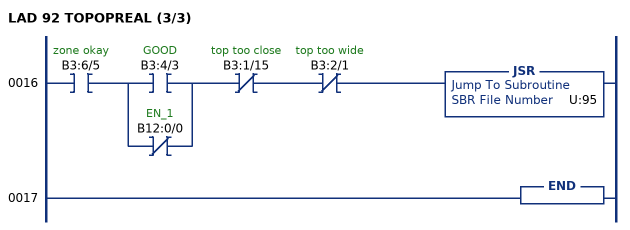
% Rung: 16 %
SOR XIC B3:6/5 BST XIC B3:4/3 NXB XIO B12:0/0 BND XIO B3:1/15 XIO B3:2/1 JSR U:95 EOR
%   B3:6/5  "zone okay" %
%   B3:4/3  GOOD %
%   B12:0/0  EN_1 %
%   B3:1/15  "top too close" %
%   B3:2/1  "top too wide" %
% Rung: 17 %
SOR END EOR

LADDER 93 "TOPOPTEST"
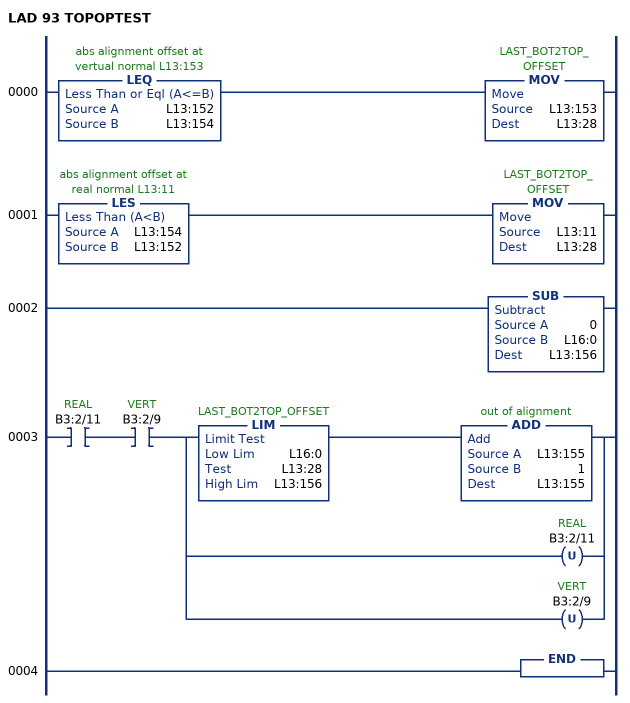
% Rung: 0 %
SOR LEQ L13:152 L13:154 MOV L13:153 L13:28 EOR
%   L13:152  "abs alignment offset at vertual normal L13:153" %
%   L13:154  "abs alignment offset at real normal L13:11" %
%   L13:153  "normal alignment offset at vertual abs L13:152" %
%   L13:28  LAST_BOT2TOP_OFFSET %
% Rung: 1 %
SOR LES L13:154 L13:152 MOV L13:11 L13:28 EOR
%   L13:154  "abs alignment offset at real normal L13:11" %
%   L13:152  "abs alignment offset at vertual normal L13:153" %
%   L13:11  "normal alignment offset at real abs L13:154" %
%   L13:28  LAST_BOT2TOP_OFFSET %
% Rung: 2 %
SOR SUB 0 L16:0 L13:156 EOR
%   L16:0  MAX_OFFSET %
% Rung: 3 %
SOR XIC B3:2/11 XIC B3:2/9 BST LIM L16:0 L13:28 L13:156 ADD L13:155 1 L13:155 NXB OTU B3:2/11 NXB OTU B3:2/9 BND EOR
%   B3:2/11  REAL %
%   B3:2/9  VERT %
%   L16:0  MAX_OFFSET %
%   L13:28  LAST_BOT2TOP_OFFSET %
%   L13:155  "out of alignment" %
% Rung: 4 %
SOR END EOR

LADDER 94 "TOPOPRANGE"
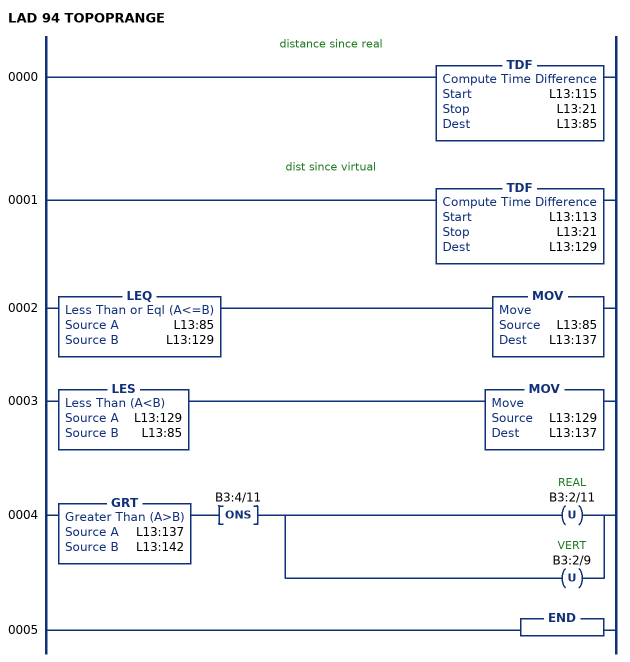
% Rung: 0 %
% distance since real %
SOR TDF L13:115 L13:21 L13:85 EOR
%   L13:115  TRAILING_EDGE_RAW  "top optic trailing edge position" %
%   L13:21  TOP_POSITION %
% Rung: 1 %
% dist since virtual %
SOR TDF L13:113 L13:21 L13:129 EOR
%   L13:113  VERTUAL_PT_RAW_CL  "virtual part center line transfer from the bottom in raw position" %
%   L13:21  TOP_POSITION %
% Rung: 2 %
SOR LEQ L13:85 L13:129 MOV L13:85 L13:137 EOR
% Rung: 3 %
SOR LES L13:129 L13:85 MOV L13:129 L13:137 EOR
% Rung: 4 %
SOR GRT L13:137 L13:142 ONS B3:4/11 BST OTU B3:2/11 NXB OTU B3:2/9 BND EOR
%   L13:142  LAST_ALIGNMENT_FAILS %
%   B3:2/11  REAL %
%   B3:2/9  VERT %
% Rung: 5 %
SOR END EOR

LADDER 95 "TOPOPOKAY"
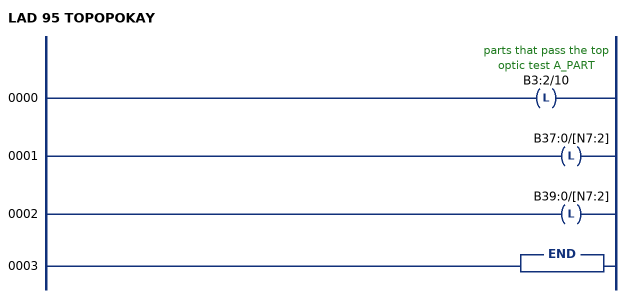
% Rung: 0 %
SOR OTL B3:2/10 EOR
%   B3:2/10  A_PART  "parts that pass the top optic test" %
% Rung: 1 %
SOR OTL B37:0/[N7:2] EOR
%   B37:0  TOP_GOOD %
%   N7:2  TOP_OPTIC_LOAD_LOC  "part load location" %
% Rung: 2 %
SOR OTL B39:0/[N7:2] EOR
%   B39:0  EX2_GOOD %
%   N7:2  TOP_OPTIC_LOAD_LOC  "part load location" %
% Rung: 3 %
SOR END EOR

LADDER 100 "1 INS5"
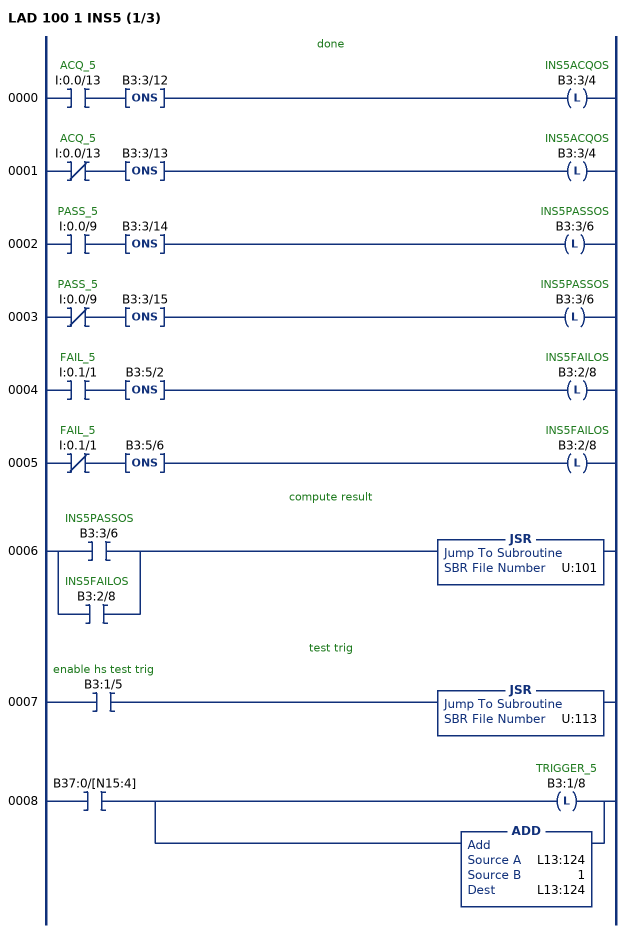
% Rung: 0 %
% done %
SOR XIC I:0.0/13 ONS B3:3/12 OTL B3:3/4 EOR
%   I:0.0/13  ACQ_5 %
%   B3:3/4  INS5ACQOS %
% Rung: 1 %
SOR XIO I:0.0/13 ONS B3:3/13 OTL B3:3/4 EOR
%   I:0.0/13  ACQ_5 %
%   B3:3/4  INS5ACQOS %
% Rung: 2 %
SOR XIC I:0.0/9 ONS B3:3/14 OTL B3:3/6 EOR
%   I:0.0/9  PASS_5 %
%   B3:3/6  INS5PASSOS %
% Rung: 3 %
SOR XIO I:0.0/9 ONS B3:3/15 OTL B3:3/6 EOR
%   I:0.0/9  PASS_5 %
%   B3:3/6  INS5PASSOS %
% Rung: 4 %
SOR XIC I:0.1/1 ONS B3:5/2 OTL B3:2/8 EOR
%   I:0.1/1  FAIL_5 %
%   B3:2/8  INS5FAILOS %
% Rung: 5 %
SOR XIO I:0.1/1 ONS B3:5/6 OTL B3:2/8 EOR
%   I:0.1/1  FAIL_5 %
%   B3:2/8  INS5FAILOS %
% Rung: 6 %
% compute result %
SOR BST XIC B3:3/6 NXB XIC B3:2/8 BND JSR U:101 EOR
%   B3:3/6  INS5PASSOS %
%   B3:2/8  INS5FAILOS %
% Rung: 7 %
% test trig %
SOR XIC B3:1/5 JSR U:113 EOR
%   B3:1/5  "enable hs test trig" %
% Rung: 8 %
SOR XIC B37:0/[N15:4] BST OTL B3:1/8 NXB ADD L13:124 1 L13:124 BND EOR
%   B37:0  TOP_GOOD %
%   N15:4  INS_5_TRIG_LOC %
%   B3:1/8  TRIGGER_5 %

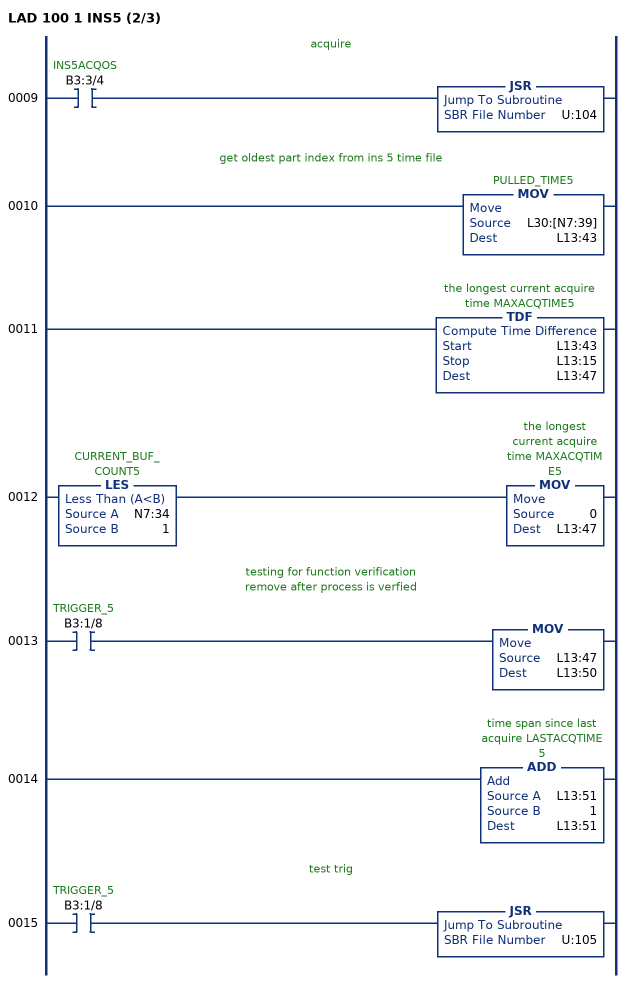
% Rung: 9 %
% acquire %
SOR XIC B3:3/4 JSR U:104 EOR
%   B3:3/4  INS5ACQOS %
% Rung: 10 %
% get oldest part index from ins 5 time file %
SOR MOV L30:[N7:39] L13:43 EOR
%   N7:39  OLDEST_PART_INDEX5 %
%   L13:43  PULLED_TIME5 %
% Rung: 11 %
SOR TDF L13:43 L13:15 L13:47 EOR
%   L13:43  PULLED_TIME5 %
%   L13:15  THE_TIME %
%   L13:47  MAXACQTIME5  "the longest current acquire time" %
% Rung: 12 %
SOR LES N7:34 1 MOV 0 L13:47 EOR
%   N7:34  CURRENT_BUF_COUNT5 %
%   L13:47  MAXACQTIME5  "the longest current acquire time" %
% Rung: 13 %
% testing for function verification
% remove after process is verfied %
SOR XIC B3:1/8 MOV L13:47 L13:50 EOR
%   B3:1/8  TRIGGER_5 %
%   L13:47  MAXACQTIME5  "the longest current acquire time" %
% Rung: 14 %
SOR ADD L13:51 1 L13:51 EOR
%   L13:51  LASTACQTIME5  "time span since last acquire" %
% Rung: 15 %
% test trig %
SOR XIC B3:1/8 JSR U:105 EOR
%   B3:1/8  TRIGGER_5 %

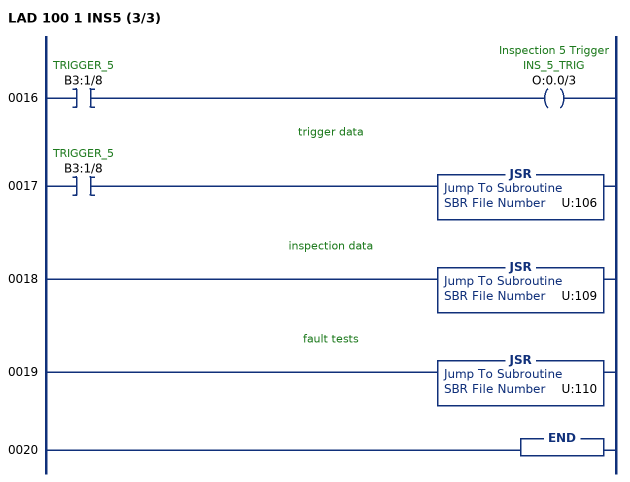
% Rung: 16 %
SOR XIC B3:1/8 OTE O:0.0/3 EOR
%   B3:1/8  TRIGGER_5 %
%   O:0.0/3  INS_5_TRIG  "Inspection 5 Trigger" %
% Rung: 17 %
% trigger data %
SOR XIC B3:1/8 JSR U:106 EOR
%   B3:1/8  TRIGGER_5 %
% Rung: 18 %
% inspection data %
SOR JSR U:109 EOR
% Rung: 19 %
% fault tests %
SOR JSR U:110 EOR
% Rung: 20 %
SOR END EOR

LADDER 101 "2 INS5RESU"
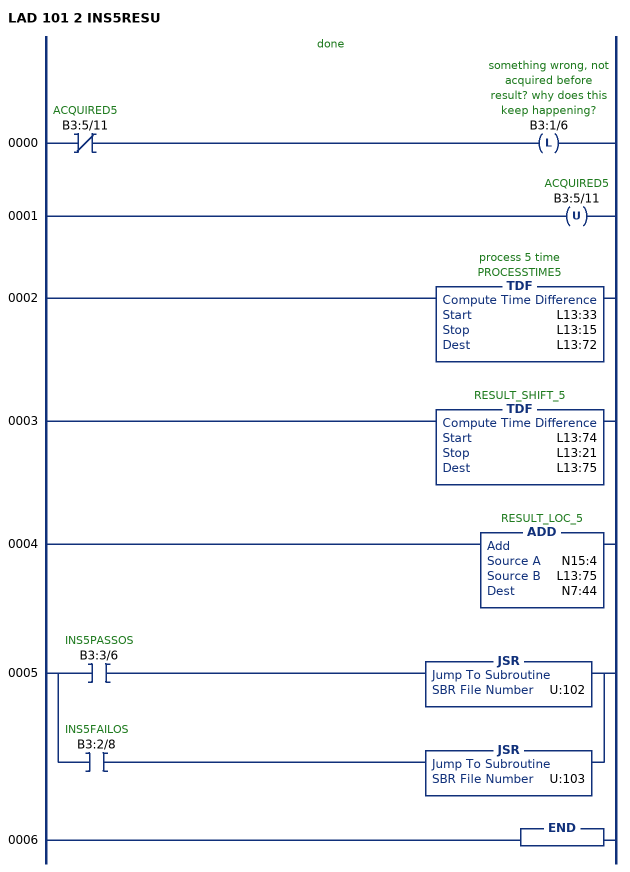
% Rung: 0 %
% done %
SOR XIO B3:5/11 OTL B3:1/6 EOR
%   B3:5/11  ACQUIRED5 %
%   B3:1/6  "something wrong, not acquired before result? why does this keep happening?" %
% Rung: 1 %
SOR OTU B3:5/11 EOR
%   B3:5/11  ACQUIRED5 %
% Rung: 2 %
SOR TDF L13:33 L13:15 L13:72 EOR
%   L13:33  TIMEOFACQ5  "the time of the last acquire" %
%   L13:15  THE_TIME %
%   L13:72  PROCESSTIME5  "process 5 time" %
% Rung: 3 %
SOR TDF L13:74 L13:21 L13:75 EOR
%   L13:74  PROCESS_START_POS_5 %
%   L13:21  TOP_POSITION %
%   L13:75  RESULT_SHIFT_5 %
% Rung: 4 %
SOR ADD N15:4 L13:75 N7:44 EOR
%   N15:4  INS_5_TRIG_LOC %
%   L13:75  RESULT_SHIFT_5 %
%   N7:44  RESULT_LOC_5 %
% Rung: 5 %
SOR BST XIC B3:3/6 JSR U:102 NXB XIC B3:2/8 JSR U:103 BND EOR
%   B3:3/6  INS5PASSOS %
%   B3:2/8  INS5FAILOS %
% Rung: 6 %
SOR END EOR

LADDER 102 "3 INS5PASS"
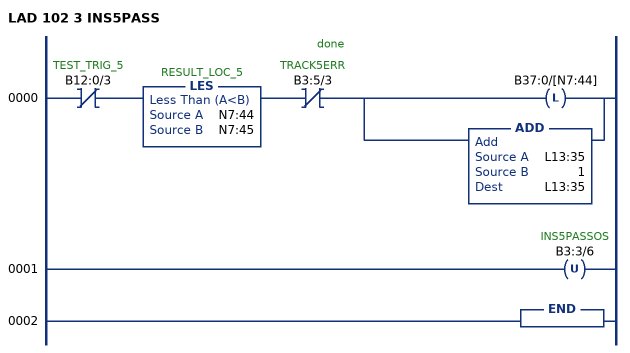
% Rung: 0 %
% done %
SOR XIO B12:0/3 LES N7:44 N7:45 XIO B3:5/3 BST OTL B37:0/[N7:44] NXB ADD L13:35 1 L13:35 BND EOR
%   B12:0/3  TEST_TRIG_5 %
%   N7:44  RESULT_LOC_5 %
%   N7:45  INS5_MAX_SHIFT  "ins 5 maximum result location" %
%   B3:5/3  TRACK5ERR %
%   B37:0  TOP_GOOD %
% Rung: 1 %
SOR OTU B3:3/6 EOR
%   B3:3/6  INS5PASSOS %
% Rung: 2 %
SOR END EOR

LADDER 103 "4 INS5FAIL"
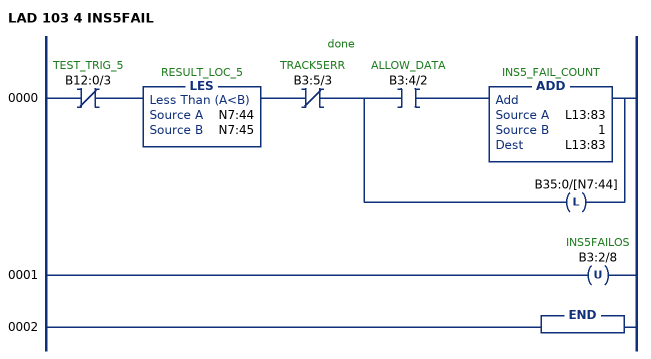
% Rung: 0 %
% done %
SOR XIO B12:0/3 LES N7:44 N7:45 XIO B3:5/3 BST XIC B3:4/2 ADD L13:83 1 L13:83 NXB OTL B35:0/[N7:44] BND EOR
%   B12:0/3  TEST_TRIG_5 %
%   N7:44  RESULT_LOC_5 %
%   N7:45  INS5_MAX_SHIFT  "ins 5 maximum result location" %
%   B3:5/3  TRACK5ERR %
%   B3:4/2  ALLOW_DATA %
%   L13:83  INS5_FAIL_COUNT %
%   B35:0  TOP_NG %
% Rung: 1 %
SOR OTU B3:2/8 EOR
%   B3:2/8  INS5FAILOS %
% Rung: 2 %
SOR END EOR

LADDER 104 "5 INS5ACQ"
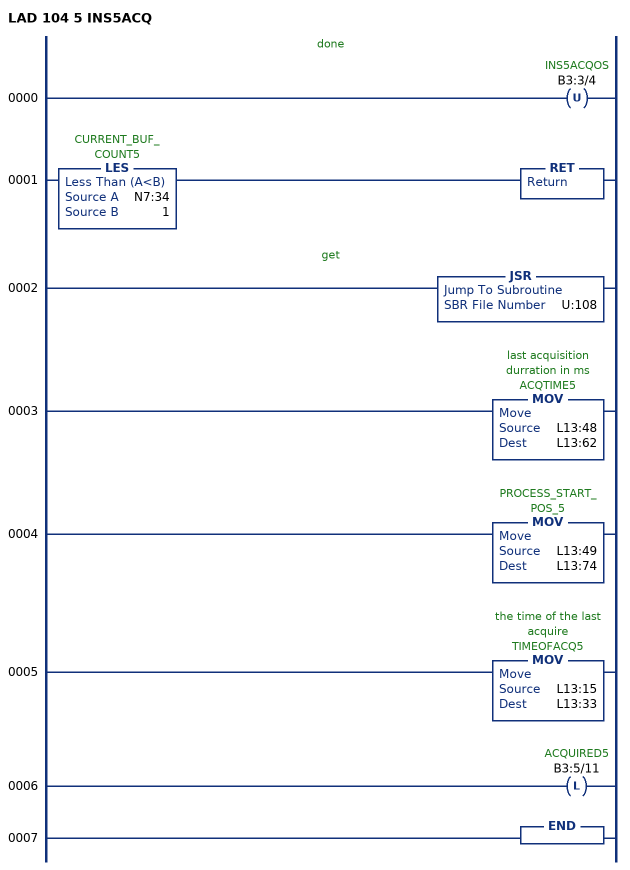
% Rung: 0 %
% done %
SOR OTU B3:3/4 EOR
%   B3:3/4  INS5ACQOS %
% Rung: 1 %
SOR LES N7:34 1 RET EOR
%   N7:34  CURRENT_BUF_COUNT5 %
% Rung: 2 %
% get %
SOR JSR U:108 EOR
% Rung: 3 %
SOR MOV L13:48 L13:62 EOR
%   L13:48  TIME_SPAN5 %
%   L13:62  ACQTIME5  "last acquisition durration in ms" %
% Rung: 4 %
SOR MOV L13:49 L13:74 EOR
%   L13:49  PULLED_POSITION5 %
%   L13:74  PROCESS_START_POS_5 %
% Rung: 5 %
SOR MOV L13:15 L13:33 EOR
%   L13:15  THE_TIME %
%   L13:33  TIMEOFACQ5  "the time of the last acquire" %
% Rung: 6 %
SOR OTL B3:5/11 EOR
%   B3:5/11  ACQUIRED5 %
% Rung: 7 %
SOR END EOR

LADDER 105 "6 Q5TESTTR"
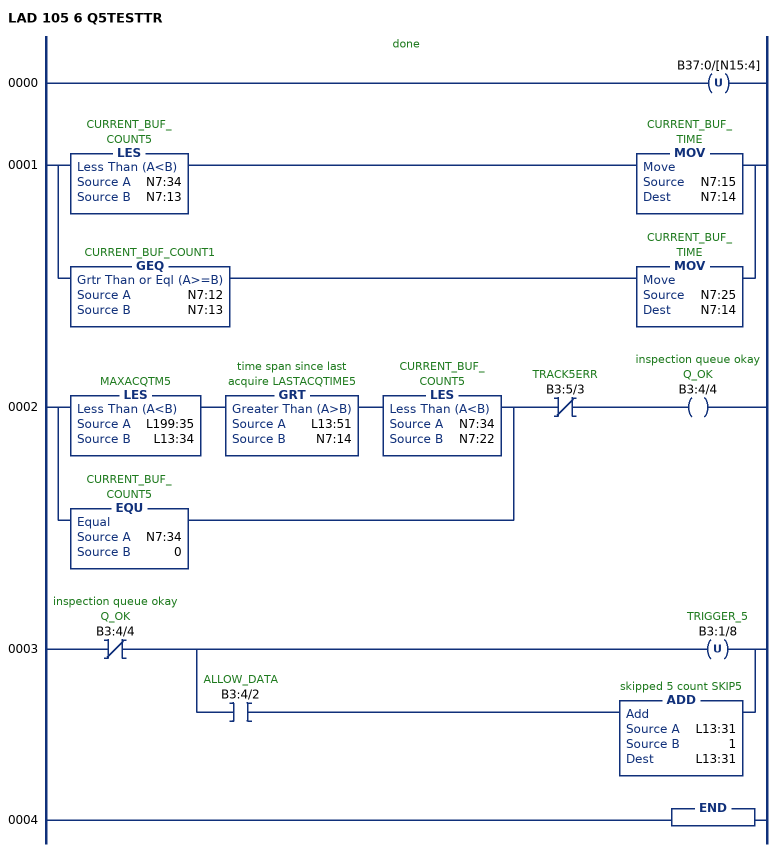
% Rung: 0 %
% done %
SOR OTU B37:0/[N15:4] EOR
%   B37:0  TOP_GOOD %
%   N15:4  INS_5_TRIG_LOC %
% Rung: 1 %
SOR BST LES N7:34 N7:13 MOV N7:15 N7:14 NXB GEQ N7:12 N7:13 MOV N7:25 N7:14 BND EOR
%   N7:34  CURRENT_BUF_COUNT5 %
%   N7:13  BUF_TRANS  "cam to pc buf transition" %
%   N7:15  CAM_BUF_TIME  "cam buf time" %
%   N7:14  CURRENT_BUF_TIME %
%   N7:12  CURRENT_BUF_COUNT1 %
%   N7:25  PC_BUF_TIME  "pc buf time" %
% Rung: 2 %
SOR BST LES L199:35 L13:34 GRT L13:51 N7:14 LES N7:34 N7:22 NXB EQU N7:34 0 BND XIO B3:5/3 OTE B3:4/4 EOR
%   L199:35  MAXACQTM5 %
%   L13:34  MAX_ACQ_ALL  "absolute max acquire time before bypass trigger" %
%   L13:51  LASTACQTIME5  "time span since last acquire" %
%   N7:14  CURRENT_BUF_TIME %
%   N7:34  CURRENT_BUF_COUNT5 %
%   N7:22  MAX_BUF_ALL  "max buffer count alowed before bypass" %
%   B3:5/3  TRACK5ERR %
%   B3:4/4  Q_OK  "inspection queue okay" %
% Rung: 3 %
SOR XIO B3:4/4 BST OTU B3:1/8 NXB XIC B3:4/2 ADD L13:31 1 L13:31 BND EOR
%   B3:4/4  Q_OK  "inspection queue okay" %
%   B3:1/8  TRIGGER_5 %
%   B3:4/2  ALLOW_DATA %
%   L13:31  SKIP5  "skipped 5 count" %
% Rung: 4 %
SOR END EOR

LADDER 106 "7 INS5TRIG"
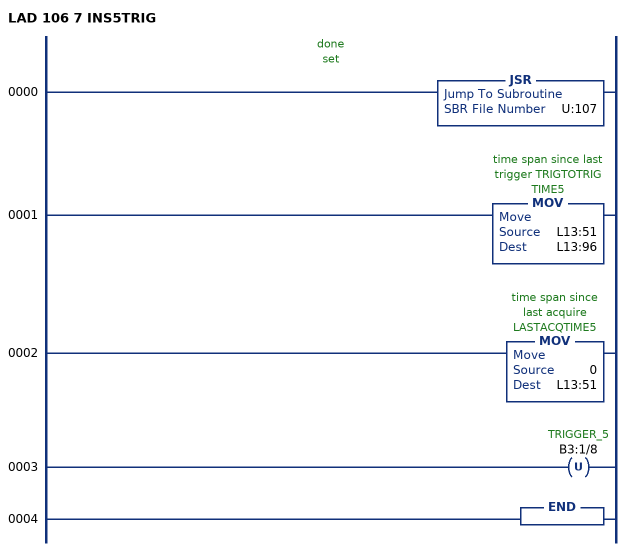
% Rung: 0 %
% done
% set %
SOR JSR U:107 EOR
% Rung: 1 %
SOR MOV L13:51 L13:96 EOR
%   L13:51  LASTACQTIME5  "time span since last acquire" %
%   L13:96  TRIGTOTRIGTIME5  "time span since last trigger" %
% Rung: 2 %
SOR MOV 0 L13:51 EOR
%   L13:51  LASTACQTIME5  "time span since last acquire" %
% Rung: 3 %
SOR OTU B3:1/8 EOR
%   B3:1/8  TRIGGER_5 %
% Rung: 4 %
SOR END EOR

LADDER 107 "8 FIFO5SET"
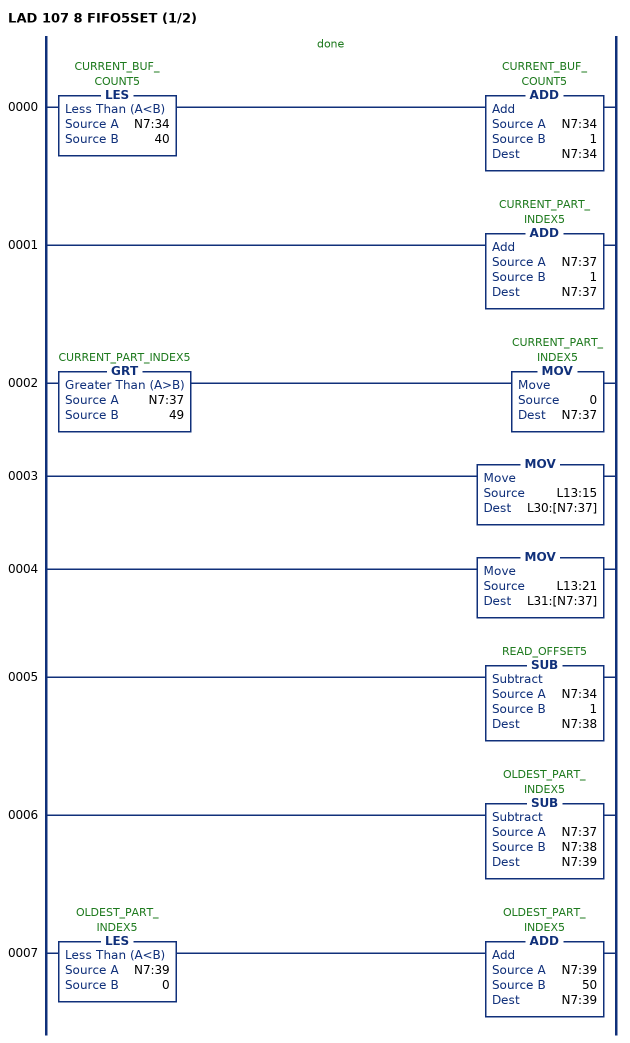
% Rung: 0 %
% done %
SOR LES N7:34 40 ADD N7:34 1 N7:34 EOR
%   N7:34  CURRENT_BUF_COUNT5 %
% Rung: 1 %
SOR ADD N7:37 1 N7:37 EOR
%   N7:37  CURRENT_PART_INDEX5 %
% Rung: 2 %
SOR GRT N7:37 49 MOV 0 N7:37 EOR
%   N7:37  CURRENT_PART_INDEX5 %
% Rung: 3 %
SOR MOV L13:15 L30:[N7:37] EOR
%   L13:15  THE_TIME %
%   N7:37  CURRENT_PART_INDEX5 %
% Rung: 4 %
SOR MOV L13:21 L31:[N7:37] EOR
%   L13:21  TOP_POSITION %
%   N7:37  CURRENT_PART_INDEX5 %
% Rung: 5 %
SOR SUB N7:34 1 N7:38 EOR
%   N7:34  CURRENT_BUF_COUNT5 %
%   N7:38  READ_OFFSET5 %
% Rung: 6 %
SOR SUB N7:37 N7:38 N7:39 EOR
%   N7:37  CURRENT_PART_INDEX5 %
%   N7:38  READ_OFFSET5 %
%   N7:39  OLDEST_PART_INDEX5 %
% Rung: 7 %
SOR LES N7:39 0 ADD N7:39 50 N7:39 EOR
%   N7:39  OLDEST_PART_INDEX5 %

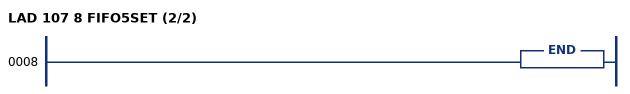
% Rung: 8 %
SOR END EOR

LADDER 108 "9 FIFO5GET"
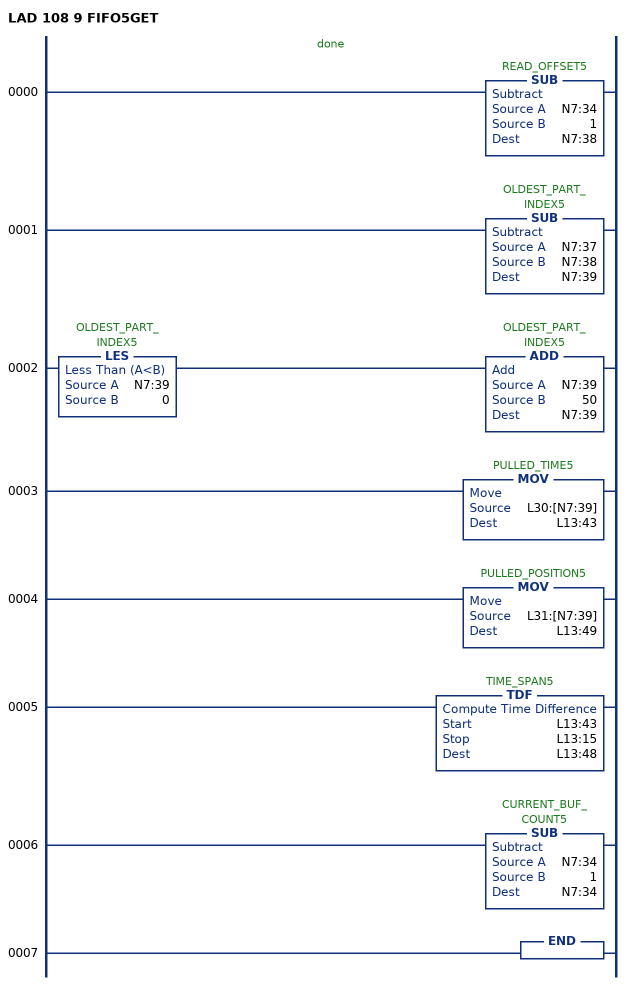
% Rung: 0 %
% done %
SOR SUB N7:34 1 N7:38 EOR
%   N7:34  CURRENT_BUF_COUNT5 %
%   N7:38  READ_OFFSET5 %
% Rung: 1 %
SOR SUB N7:37 N7:38 N7:39 EOR
%   N7:37  CURRENT_PART_INDEX5 %
%   N7:38  READ_OFFSET5 %
%   N7:39  OLDEST_PART_INDEX5 %
% Rung: 2 %
SOR LES N7:39 0 ADD N7:39 50 N7:39 EOR
%   N7:39  OLDEST_PART_INDEX5 %
% Rung: 3 %
SOR MOV L30:[N7:39] L13:43 EOR
%   N7:39  OLDEST_PART_INDEX5 %
%   L13:43  PULLED_TIME5 %
% Rung: 4 %
SOR MOV L31:[N7:39] L13:49 EOR
%   N7:39  OLDEST_PART_INDEX5 %
%   L13:49  PULLED_POSITION5 %
% Rung: 5 %
SOR TDF L13:43 L13:15 L13:48 EOR
%   L13:43  PULLED_TIME5 %
%   L13:15  THE_TIME %
%   L13:48  TIME_SPAN5 %
% Rung: 6 %
SOR SUB N7:34 1 N7:34 EOR
%   N7:34  CURRENT_BUF_COUNT5 %
% Rung: 7 %
SOR END EOR

LADDER 109 "10INSDATA5"
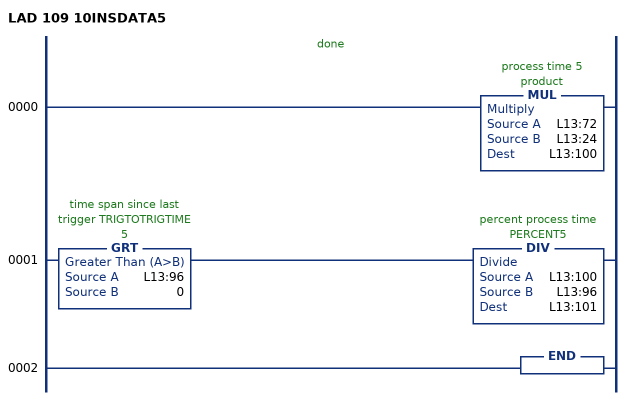
% Rung: 0 %
% done %
SOR MUL L13:72 L13:24 L13:100 EOR
%   L13:72  PROCESSTIME5  "process 5 time" %
%   L13:24  "multiplyer to make devision come out to a percentage" %
%   L13:100  "process time 5 product" %
% Rung: 1 %
SOR GRT L13:96 0 DIV L13:100 L13:96 L13:101 EOR
%   L13:96  TRIGTOTRIGTIME5  "time span since last trigger" %
%   L13:100  "process time 5 product" %
%   L13:101  PERCENT5  "percent process time" %
% Rung: 2 %
SOR END EOR

LADDER 110 "11TSTFALT5"
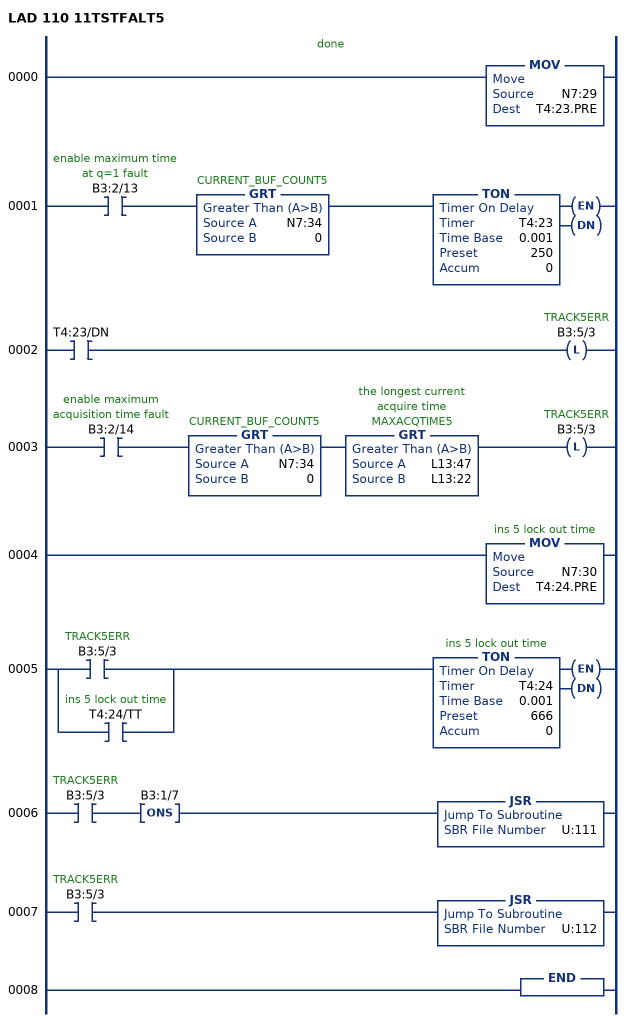
% Rung: 0 %
% done %
SOR MOV N7:29 T4:23.PRE EOR
%   N7:29  "max allowed ms time for q to be above 1 if safe fault is used" %
% Rung: 1 %
SOR XIC B3:2/13 GRT N7:34 0 TON T4:23 0.001 250 0 EOR
%   B3:2/13  "enable maximum time at q=1 fault" %
%   N7:34  CURRENT_BUF_COUNT5 %
% Rung: 2 %
SOR XIC T4:23/DN OTL B3:5/3 EOR
%   B3:5/3  TRACK5ERR %
% Rung: 3 %
SOR XIC B3:2/14 GRT N7:34 0 GRT L13:47 L13:22 OTL B3:5/3 EOR
%   B3:2/14  "enable maximum acquisition time fault" %
%   N7:34  CURRENT_BUF_COUNT5 %
%   L13:47  MAXACQTIME5  "the longest current acquire time" %
%   L13:22  "maximum of the longest acquire time allowed if maximum acquire time fault is enabled" %
%   B3:5/3  TRACK5ERR %
% Rung: 4 %
SOR MOV N7:30 T4:24.PRE EOR
%   N7:30  "ms time setting to lock out inspection to give all pending images a chance to clear" %
%   T4:24  "ins 5 lock out time" %
% Rung: 5 %
SOR BST XIC B3:5/3 NXB XIC T4:24/TT BND TON T4:24 0.001 666 0 EOR
%   B3:5/3  TRACK5ERR %
%   T4:24  "ins 5 lock out time" %
% Rung: 6 %
SOR XIC B3:5/3 ONS B3:1/7 JSR U:111 EOR
%   B3:5/3  TRACK5ERR %
% Rung: 7 %
SOR XIC B3:5/3 JSR U:112 EOR
%   B3:5/3  TRACK5ERR %
% Rung: 8 %
SOR END EOR

LADDER 111 "12INS5FIX1"
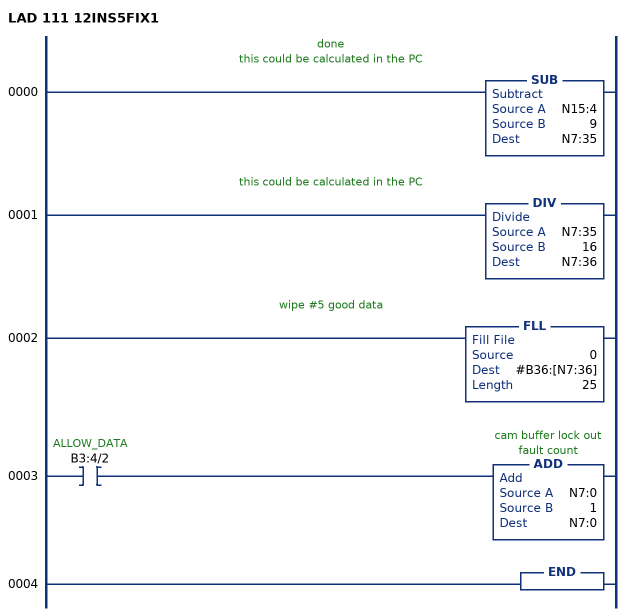
% Rung: 0 %
% done
% this could be calculated in the PC %
SOR SUB N15:4 9 N7:35 EOR
%   N15:4  INS_5_TRIG_LOC %
% Rung: 1 %
% this could be calculated in the PC %
SOR DIV N7:35 16 N7:36 EOR
% Rung: 2 %
% wipe #5 good data %
SOR FLL 0 #B36:[N7:36] 25 EOR
% Rung: 3 %
SOR XIC B3:4/2 ADD N7:0 1 N7:0 EOR
%   B3:4/2  ALLOW_DATA %
%   N7:0  "cam buffer lock out fault count" %
% Rung: 4 %
SOR END EOR

LADDER 112 "13INS5FIX2"
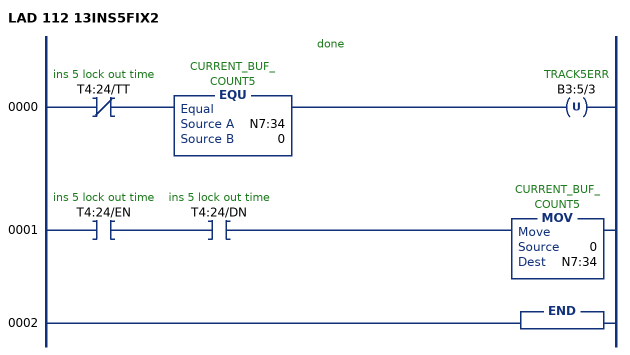
% Rung: 0 %
% done %
SOR XIO T4:24/TT EQU N7:34 0 OTU B3:5/3 EOR
%   T4:24  "ins 5 lock out time" %
%   N7:34  CURRENT_BUF_COUNT5 %
%   B3:5/3  TRACK5ERR %
% Rung: 1 %
SOR XIC T4:24/EN XIC T4:24/DN MOV 0 N7:34 EOR
%   T4:24  "ins 5 lock out time" %
%   N7:34  CURRENT_BUF_COUNT5 %
% Rung: 2 %
SOR END EOR

LADDER 113 "14 HSTRIG5"
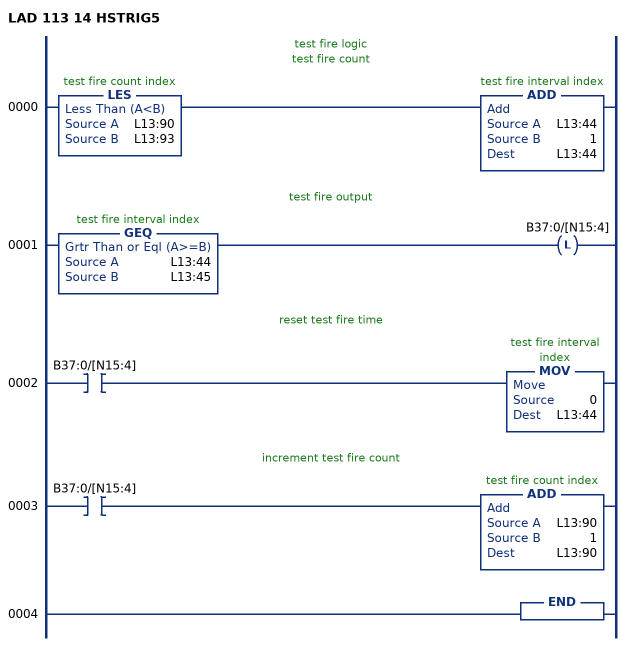
% Rung: 0 %
% test fire logic
% 
% test fire count %
SOR LES L13:90 L13:93 ADD L13:44 1 L13:44 EOR
%   L13:90  "test fire count index" %
%   L13:93  "test fire count" %
%   L13:44  "test fire interval index" %
% Rung: 1 %
% test fire output %
SOR GEQ L13:44 L13:45 OTL B37:0/[N15:4] EOR
%   L13:44  "test fire interval index" %
%   L13:45  "test fire interval" %
%   B37:0  TOP_GOOD %
%   N15:4  INS_5_TRIG_LOC %
% Rung: 2 %
% reset test fire time %
SOR XIC B37:0/[N15:4] MOV 0 L13:44 EOR
%   B37:0  TOP_GOOD %
%   N15:4  INS_5_TRIG_LOC %
%   L13:44  "test fire interval index" %
% Rung: 3 %
% increment test fire count %
SOR XIC B37:0/[N15:4] ADD L13:90 1 L13:90 EOR
%   B37:0  TOP_GOOD %
%   N15:4  INS_5_TRIG_LOC %
%   L13:90  "test fire count index" %
% Rung: 4 %
SOR END EOR

LADDER 120 "1 INS6"
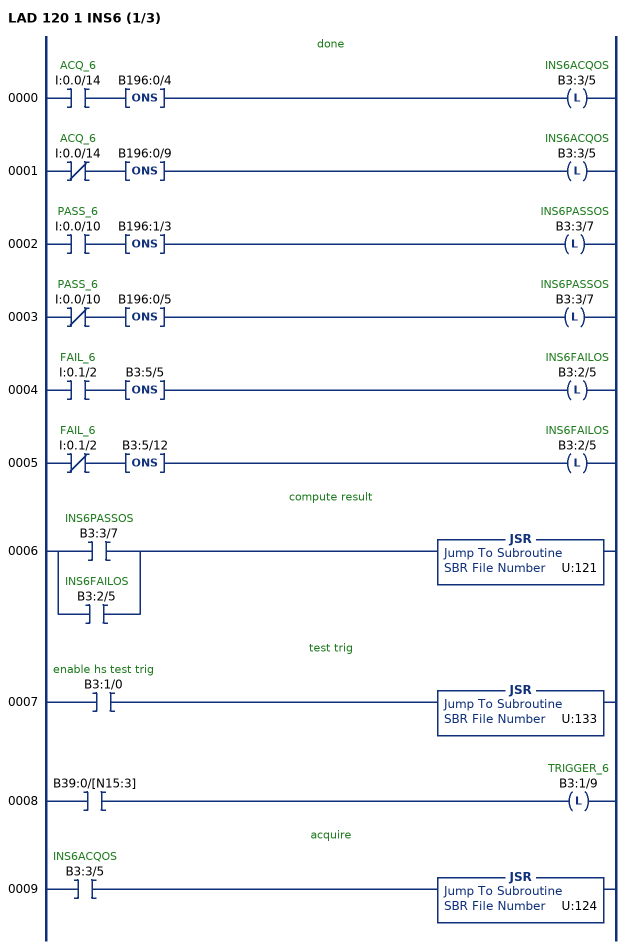
% Rung: 0 %
% done %
SOR XIC I:0.0/14 ONS B196:0/4 OTL B3:3/5 EOR
%   I:0.0/14  ACQ_6 %
%   B3:3/5  INS6ACQOS %
% Rung: 1 %
SOR XIO I:0.0/14 ONS B196:0/9 OTL B3:3/5 EOR
%   I:0.0/14  ACQ_6 %
%   B3:3/5  INS6ACQOS %
% Rung: 2 %
SOR XIC I:0.0/10 ONS B196:1/3 OTL B3:3/7 EOR
%   I:0.0/10  PASS_6 %
%   B3:3/7  INS6PASSOS %
% Rung: 3 %
SOR XIO I:0.0/10 ONS B196:0/5 OTL B3:3/7 EOR
%   I:0.0/10  PASS_6 %
%   B3:3/7  INS6PASSOS %
% Rung: 4 %
SOR XIC I:0.1/2 ONS B3:5/5 OTL B3:2/5 EOR
%   I:0.1/2  FAIL_6 %
%   B3:2/5  INS6FAILOS %
% Rung: 5 %
SOR XIO I:0.1/2 ONS B3:5/12 OTL B3:2/5 EOR
%   I:0.1/2  FAIL_6 %
%   B3:2/5  INS6FAILOS %
% Rung: 6 %
% compute result %
SOR BST XIC B3:3/7 NXB XIC B3:2/5 BND JSR U:121 EOR
%   B3:3/7  INS6PASSOS %
%   B3:2/5  INS6FAILOS %
% Rung: 7 %
% test trig %
SOR XIC B3:1/0 JSR U:133 EOR
%   B3:1/0  "enable hs test trig" %
% Rung: 8 %
SOR XIC B39:0/[N15:3] OTL B3:1/9 EOR
%   B39:0  EX2_GOOD %
%   N15:3  INS_6_TRIG_LOC %
%   B3:1/9  TRIGGER_6 %
% Rung: 9 %
% acquire %
SOR XIC B3:3/5 JSR U:124 EOR
%   B3:3/5  INS6ACQOS %

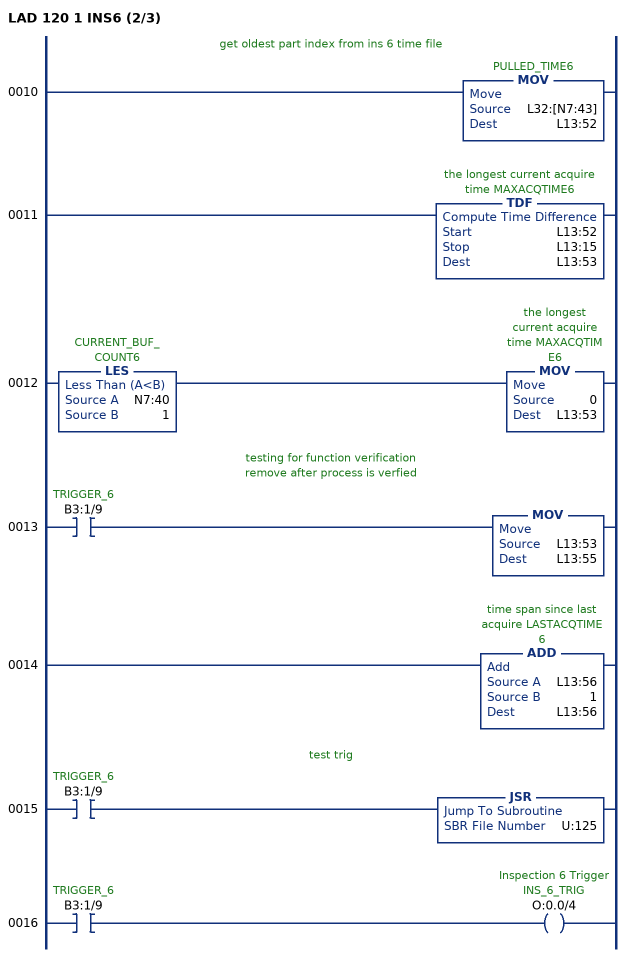
% Rung: 10 %
% get oldest part index from ins 6 time file %
SOR MOV L32:[N7:43] L13:52 EOR
%   N7:43  OLDEST_PART_INDEX6 %
%   L13:52  PULLED_TIME6 %
% Rung: 11 %
SOR TDF L13:52 L13:15 L13:53 EOR
%   L13:52  PULLED_TIME6 %
%   L13:15  THE_TIME %
%   L13:53  MAXACQTIME6  "the longest current acquire time" %
% Rung: 12 %
SOR LES N7:40 1 MOV 0 L13:53 EOR
%   N7:40  CURRENT_BUF_COUNT6 %
%   L13:53  MAXACQTIME6  "the longest current acquire time" %
% Rung: 13 %
% testing for function verification
% remove after process is verfied %
SOR XIC B3:1/9 MOV L13:53 L13:55 EOR
%   B3:1/9  TRIGGER_6 %
%   L13:53  MAXACQTIME6  "the longest current acquire time" %
% Rung: 14 %
SOR ADD L13:56 1 L13:56 EOR
%   L13:56  LASTACQTIME6  "time span since last acquire" %
% Rung: 15 %
% test trig %
SOR XIC B3:1/9 JSR U:125 EOR
%   B3:1/9  TRIGGER_6 %
% Rung: 16 %
SOR XIC B3:1/9 OTE O:0.0/4 EOR
%   B3:1/9  TRIGGER_6 %
%   O:0.0/4  INS_6_TRIG  "Inspection 6 Trigger" %

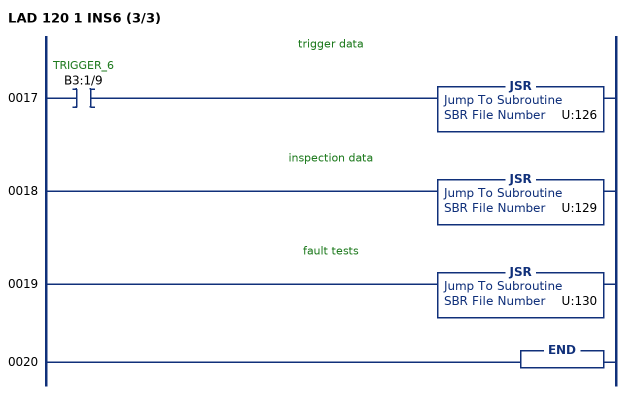
% Rung: 17 %
% trigger data %
SOR XIC B3:1/9 JSR U:126 EOR
%   B3:1/9  TRIGGER_6 %
% Rung: 18 %
% inspection data %
SOR JSR U:129 EOR
% Rung: 19 %
% fault tests %
SOR JSR U:130 EOR
% Rung: 20 %
SOR END EOR

LADDER 121 "2 INS6RESU"
